FUNCTION_BLOCK FB_NciChannelTangential_Test EXTENDS TcUnit.FB_TestSuite
VAR
    ChannelTan  : FB_NciChannelTangential;
    DummyTable  : ST_NciFeedGroupTable;
END_VAR

Test_StartFeedTable_ResetsDoneFlags();
Test_ResetChannel_ClearsErrors();
Test_BuildExtGroup_ClearsGroupedFlag();

METHOD Test_BuildExtGroup_ClearsGroupedFlag
VAR_INST
END_VAR
TEST('Test_BuildExtGroup_ClearsGroupedFlag');

// ACT - Budowanie grupy zawierającej dodatkowo oś Q1
ChannelTan.BuildGroup();

// ASSERT
AssertFalse(Condition := ChannelTan.IsGrouped,
            Message := 'IsGrouped nie zostalo zresetowane przy wywolaniu BuildGroup na EXT grupie!');
AssertFalse(Condition := ChannelTan.ChannelError,
            Message := 'Bledy kanalu tangencjalnego nie zostaly zresetowane przy probie BuildGroup!');

TEST_FINISHED();
END_METHOD

METHOD Test_ResetChannel_ClearsErrors
VAR_INST
END_VAR
TEST('Test_ResetChannel_ClearsErrors');

// ACT
ChannelTan.ResetChannel();

// ASSERT
AssertFalse(Condition := ChannelTan.ChannelError,
            Message := 'Flaga bledu kanalu tangencjalnego nie zniknela po wywolaniu ResetChannel!');
AssertEquals_UDINT(Expected := 0, 
                   Actual := ChannelTan.ChannelErrorId, 
                   Message := 'ID bledu nie zostalo wyzerowane w kanale tangencjalnym!');

TEST_FINISHED();
END_METHOD

METHOD Test_StartFeedTable_ResetsDoneFlags
VAR_INST
END_VAR
TEST('Test_StartFeedTable_ResetsDoneFlags');

// ACT - Przekazujemy strukturę z tabelą i startujemy feedowanie punktów
ChannelTan.StartFeedTable(stTable := DummyTable);

// ASSERT - Flagi końca powinny być natychmiast wyzerowane
AssertFalse(Condition := ChannelTan.IsFeedingDone,
            Message := 'IsFeedingDone powinno byc FALSE na starcie interpolacji tabelarycznej!');
AssertFalse(Condition := ChannelTan.IsChannelDone,
            Message := 'IsChannelDone powinno byc FALSE na starcie interpolacji tabelarycznej!');

TEST_FINISHED();
END_METHOD

END_FUNCTION_BLOCK

(* stored: Version 1.1.0.1, ProductVersion 3.1.4024.15
   POU FB_NciChannelTangential_Test: Id {b1b2c3d4-e5f6-4789-9999-000000000001}, SpecialFunc None
   Method Test_BuildExtGroup_ClearsGroupedFlag: Id {b1b2c3d4-e5f6-4789-9999-000000000004}
   Method Test_ResetChannel_ClearsErrors: Id {b1b2c3d4-e5f6-4789-9999-000000000003}
   Method Test_StartFeedTable_ResetsDoneFlags: Id {b1b2c3d4-e5f6-4789-9999-000000000002} *)
